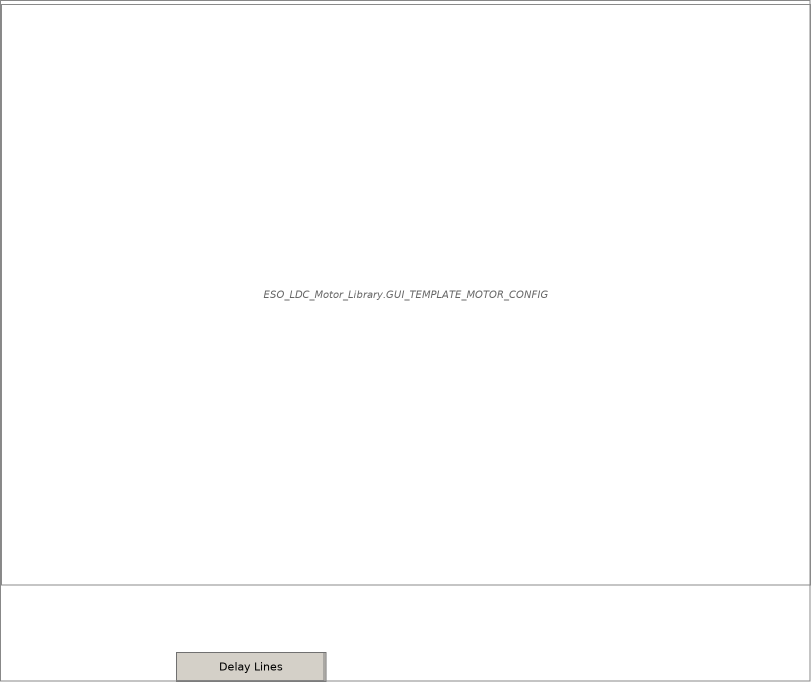
VISUALIZATION DL_MOTOR_01_CONFIG  // 811x682
    Frame (1,4 810x581)
        shows ESO_LDC_Motor_Library.GUI_TEMPLATE_MOTOR_CONFIG(m_Instance := MAIN.DL_Motor_01)
    Button (176,652 150x30), "Delay Lines"
        OnMouseDown: change screen: SCIFY_Delay_Lines
END_VISUALIZATION

(* stored: Version 1.1.0.1, ProductVersion 3.1.4024.12
   Visu DL_MOTOR_01_CONFIG: Id {35ff1947-087e-4c9f-b8c1-44384f22caaa} *)
